// TwinCAT 3 PLC project MaterialHandling
// ProgramVersion: 3.1.4026.20
// CompilerDefines: VISU_USEPROPERTYINFO
// libraries:
//   Tc2_Standard, * (Beckhoff Automation GmbH)
//   Tc2_System, * (Beckhoff Automation GmbH)
// project tree:
//   Class Diagram/ Code Design Architecture.TcCD (not stored)
//   DUTs/ E_AutoState.TcDUT, E_ErrorHandling.TcDUT, E_Mode.TcDUT
//   / GlobalTextList.TcGTLO, PlcTask.TcTTO, Visualization Manager.TcVMO (not stored)
//   GVLs/ IOs.TcGVL
//   POUs/ FB_ErrorHandling.TcPOU, FB_AutoState.TcPOU, FB_ModeManager.TcPOU, MAIN.TcPOU, FB_StateMachine.TcPOU
//   VISUs/ Visualization.TcVIS
// real-time tasks:
//   TASK PlcTask: cycle T#10ms, priority 20, ADS port 350

CONFIGURATION MaterialHandling
    RESOURCE PLC ON TwinCAT3
        TASK PlcTask(INTERVAL := T#10ms, PRIORITY := 20);
        PROGRAM MAIN WITH PlcTask : MAIN;
    END_RESOURCE
END_CONFIGURATION

// ---- DUTs/E_AutoState.TcDUT
{attribute 'to_string'}
TYPE E_AutoState :
(
	Create_Product:= 10,
	Load_Conveyor:= 20,
	Transfer_To_MC:= 30,
	Machine_Start:= 40,
	Wait_Machine_Busy:= 50,
	Wait_Machine_Complete:= 60,
	Exit_MC:= 70,
	MOVE_To_Unload:= 80,
	Remove_Product:= 90,
	Complete:= 100
);
END_TYPE

// ---- DUTs/E_ErrorHandling.TcDUT
{attribute 'to_string'}
TYPE E_ErrorHandling :
(
	Fault := 900,
	Emergency := 999,
	No_Error := 0
);
END_TYPE

// ---- DUTs/E_Mode.TcDUT
{attribute 'to_string'}
TYPE E_Mode :
(
	Idle := 0,
	Auto := 1,
	Manual:= 2,
	Error:= 3
);
END_TYPE

// ---- GVLs/IOs.TcGVL
{attribute 'OPC.UA.DA' := '1'}
{attribute 'OPC.UA.DA.Access' := '3'}
VAR_GLOBAL
////////////////////////////////
    //Inputs...............
////////////////////////////////
(*1*)	 xSensor_LoadStation:        BOOL;
(*2*)    xSensor_BeforeEntry:        BOOL;
(*3*)    xSensor_AtExit:             BOOL;
(*4*)    xEStop:                     BOOL;    //Stop the complete Machine
(*5*)	 xPB_ManualRun_Pressed:      BOOL;    //PB = Push Button  
(*6*)    xMC_Opened:                 BOOL;    //MC = Machine Center
(*7*)    xMC_IsBusy:                 BOOL;
(*8*)	 xMC_HasError:               BOOL;
(*9*)    xrMC_Progress:              DINT;
(*10*)   xSel_Auto:                  BOOL;
(*11*)   xSel_Manual:                BOOL;
(*12*)	 xSel_OFF:                   BOOL;

(*13*)   xSystemPower:               BOOL;    // Power System ON/OFF - Input from HMI or Scene button
(*14*)   xSystemReset:               BOOL;    // System Reset - Input from HMI or Scene button 
/////////////////////////////////
    //Outputs...............
/////////////////////////////////
(*1*)	 xEmitter:                   BOOL;
(*2*)    xConv_LoadStation:          BOOL;    //Conv = Conveyor
(*3*)    xCurvedConv_CCW:            BOOL;
(*4*)    xConv_BeforeEntry:          BOOL;    //Stop the complete Machine
(*5*)	 xMC_Start:                  BOOL;    //PB = Push Button
(*6*)    xMC_Stop:                   BOOL;    //MC = Machine Center
(*7*)    xMC_Reset:                  BOOL;
(*8*)	 xMC_ProduceLids:            BOOL;    //True: Produce Lids , False: Produce Bases
(*9*)    xConv_AfterProcess:         BOOL;
(*10*)   xRemover:                   BOOL;
(*11*)   xPb_ManualRun_Light:        BOOL;
END_VAR

// ---- POUs/MAIN.TcPOU
PROGRAM MAIN
VAR
	fbStateMachine: FB_StateMachine;
	eErrorType: E_ErrorHandling;
	xEmitter_Manual: BOOL;  //Simulation
	eMode: E_Mode;
	////// Inputs & Outputs
	xEStop: BOOL;
	xPB_ManualRun_Pressed: BOOL;
	xSel_Auto: BOOL;
    xSel_Manual: BOOL;
	///////////
	xEmitter: BOOL;
	xConv_LoadStation: BOOL;
	xCurvedConv_CCW: BOOL;
	xConv_BeforeEntry: BOOL;
	xMC_Start: BOOL;
	xMC_Stop: BOOL;
	xMC_Reset: BOOL;
	xMC_ProduceLids: BOOL;
	xConv_AfterProcess: BOOL;
	xRemover: BOOL;
END_VAR


xEStop:= NOT IOs.xEStop;
xPB_ManualRun_Pressed:= IOs.xPB_ManualRun_Pressed;
xSel_Auto:= IOs.xSel_Auto;
xSel_Manual:= IOs.xSel_Manual;

IF IOs.xSystemPower THEN
	fbStateMachine(xEmitter_Manual:= xEmitter_Manual,xESTOP:= xESTOP, xPB_ManualRun_Pressed:= xPB_ManualRun_Pressed, xSel_Auto:= xSel_Auto, xSel_Manual:= xSel_Manual);
    eMode := fbStateMachine.eMode;
    eErrorType:= fbStateMachine.eErrorType;
END_IF


IOs.xEmitter := fbStateMachine.xEmitter;
IOs.xConv_LoadStation := fbStateMachine.xConv_LoadStation;
IOs.xCurvedConv_CCW := fbStateMachine.xCurvedConv_CCW;
IOs.xConv_BeforeEntry := fbStateMachine.xConv_BeforeEntry;
IOs.xMC_Start := fbStateMachine.xMC_Start;
IOs.xMC_Stop := fbStateMachine.xMC_Stop;
IOs.xMC_Reset := fbStateMachine.xMC_Reset;
IOs.xMC_ProduceLids := fbStateMachine.xMC_ProduceLids;
IOS.xConv_AfterProcess := fbStateMachine.xConv_AfterProcess; 
IOs.xRemover := fbStateMachine.xRemover;

END_PROGRAM

// ---- POUs/FB_StateMachine.TcPOU
FUNCTION_BLOCK FB_StateMachine

VAR
	fbModeManager: FB_ModeManager;
	fbAutoState: FB_AutoState;
	xEnable_Auto: BOOL;
	xReset_Auto: BOOL;
END_VAR
VAR_INPUT
	xEmitter_Manual: BOOL;
	xEStop: BOOL;
	xPB_ManualRun_Pressed: BOOL;
	xSel_Auto: BOOL;
    xSel_Manual: BOOL;
END_VAR
VAR_OUTPUT
	eErrorType: E_ErrorHandling;
	eMode: E_Mode;
	
	xEmitter: BOOL;
	xConv_LoadStation: BOOL;
	xCurvedConv_CCW: BOOL;
	xConv_BeforeEntry: BOOL;
	xMC_Start: BOOL;
	xMC_Stop: BOOL;
	xMC_Reset: BOOL;
	xMC_ProduceLids: BOOL;
	xConv_AfterProcess: BOOL;
	xRemover: BOOL;
END_VAR

fbModeManager(xEStop := xEStop, xSel_Auto:= xSel_Auto, xSel_Manual:= xSel_Manual);
eMode := fbModeManager.eMode;
eErrorType:= fbModeManager.eErrorType;

IF eMode = Auto THEN
	xEnable_Auto := TRUE;
	xReset_Auto := FALSE;
END_IF
IF eMode = Idle OR eMode = Manual THEN
		xEnable_Auto := FALSE;
	    xReset_Auto := TRUE;
END_IF
	
 CASE eMode OF
	
	Auto:
	   
	   fbAutoState(xEnable:=xEnable_Auto, xReset:=xReset_Auto);
	   
	   xEmitter := fbAutoState.xEmitter;
       xConv_LoadStation := fbAutoState.xConv_LoadStation;
	   xCurvedConv_CCW := fbAutoState.xCurvedConv_CCW;
	   xConv_BeforeEntry := fbAutoState.xConv_BeforeEntry;
	   xMC_Start := fbAutoState.xMC_Start;
	   xMC_ProduceLids := fbAutoState.xMC_ProduceLids;
	   xConv_AfterProcess := fbAutoState.xConv_AfterProcess;
	   xRemover := fbAutoState.xRemover;
	   
	Manual:
	   
	   IF xPB_ManualRun_Pressed THEN
		   xMC_Start := xPB_ManualRun_Pressed;  //Robot in the Scene is predefined to work only when the raw material detected from the cell-Sensor; IF operator released the PB during the Transfer, it supposed to finish the current job unless he pressed Stop
           //xPb_ManualRun_Light:= TRUE;    don't forget
		   xConv_LoadStation:= TRUE;
		   xCurvedConv_CCW:= TRUE;
		   xConv_BeforeEntry:= TRUE;
		   xConv_AfterProcess:=TRUE;
		   xEmitter := xEmitter_Manual;  //Operator should feed the Material manually obe by one (Later with HMI)
		   xRemover:= TRUE;
	   END_IF
	   
	   fbAutoState(xEnable:=xEnable_Auto, xReset:=xReset_Auto);
	  	
	 Idle:
	    
	    xConv_LoadStation:= FALSE;
		xCurvedConv_CCW:= FALSE;
		xConv_BeforeEntry:= FALSE;
		xConv_AfterProcess:= FALSE;
		xMC_Start:= FALSE;
		xMC_Stop:= FALSE;
		xEmitter:= FALSE;
		xRemover:= FALSE;
		xMC_Reset:= TRUE;
		xMC_Reset:= FALSE; //Trigger once at the beginning
		
		fbAutoState(xEnable:=xEnable_Auto, xReset:=xReset_Auto);
	  
  END_CASE

END_FUNCTION_BLOCK

// ---- POUs/FB_ModeManager.TcPOU
FUNCTION_BLOCK FB_ModeManager
VAR_INPUT
	xEStop: BOOL;
	xSel_Auto: BOOL;
	xSel_Manual: BOOL;
END_VAR
VAR_OUTPUT
	eMode: E_MODE;
	eErrorType: E_ErrorHAndling;
END_VAR
VAR
	fbErrorHandling: FB_ErrorHAndling;
END_VAR

IF IOs.xMC_HasError OR xEStop THEN  //Emergency_Stop is NC designed!
	eMode:= Error;
  ELSIF IOs.xSel_Auto THEN
   eMode:= Auto;
	ELSIF IOs.xSel_Manual THEN
		eMode:= Manual;
		ELSE
			eMode:= Idle;
END_IF


fbErrorHandling(xEStop := xEStop);
eErrorType:= fbErrorHandling.eErrorHandling;

END_FUNCTION_BLOCK

// ---- POUs/FB_ErrorHandling.TcPOU
FUNCTION_BLOCK FB_ErrorHandling
VAR_INPUT
	xEStop: BOOL;
END_VAR
VAR_OUTPUT
	eErrorHandling: E_ErrorHandling;
END_VAR
VAR
END_VAR

IF xEStop THEN
	eErrorHandling:= Emergency;
ELSIF IOs.xMC_HasError THEN
		eErrorHandling:= Fault;
		ELSE
			eErrorHandling:= No_Error;
END_IF

END_FUNCTION_BLOCK

// ---- POUs/FB_AutoState.TcPOU
FUNCTION_BLOCK FB_AutoState

VAR
	eAutoState: E_AutoState := Create_Product;
	//pPointer: POINTER TO E_MODE;
END_VAR
VAR_INPUT
	xEnable: BOOL;
	xReset: BOOL;
END_VAR
VAR_OUTPUT
	xEmitter: BOOL;
	xConv_LoadStation: BOOL;
	xCurvedConv_CCW: BOOL;
	xConv_BeforeEntry: BOOL;
	xMC_Start: BOOL;
	xMC_ProduceLids: BOOL;
	xConv_AfterProcess: BOOL;
	xRemover: BOOL;
END_VAR

IF xReset THEN
	IF IOs.xSystemReset THEN  //If Operator clicked reset=> Product on conveyor has been cleared ; If Not => system will continue running same product when back to Auto 
     eAutoState:= Create_Product;
    END_IF
   ELSIF xEnable THEN	
	
CASE eAutoState OF

(*10*) Create_Product:
	
	   xEmitter:= TRUE;
	   IF IOs.xSensor_LoadStation THEN
		  eAutoState := Load_Conveyor;
	   END_IF
	
(*20*) Load_Conveyor: 
	
	   xEmitter := FALSE;
	   xConv_LoadStation:= TRUE;
	   IF NOT IOs.xSensor_LoadStation THEN
		   eAutoState:= Transfer_To_MC;
	   END_IF
 
(*30*) Transfer_To_MC: 
	
	   xCurvedConv_CCW:= TRUE;
	   xConv_BeforeEntry:= TRUE;
	   IF IOs.xSensor_BeforeEntry THEN
		   eAutoState:= Machine_Start;
	   END_IF
	   
(*40*) Machine_Start: 

       xConv_LoadStation:= FALSE;
       xCurvedConv_CCW:= FALSE;
       xMC_Start:= TRUE;
       xMC_ProduceLids:= 0; //0 Produce base
	   IF IOs.xMC_IsBusy THEN
       eAutoState:= Wait_Machine_Busy;
	   END_IF
	   
(*50*) Wait_Machine_Busy: 
	 
	    xConv_BeforeEntry:= FALSE;
		IF (IOs.xrMC_Progress > 0) AND (IOs.xrMC_Progress < 100) THEN
		eAutoState:= Wait_Machine_Complete;
	    END_IF
	 
(*60*) Wait_Machine_Complete:  
	   
	   xMC_Start:= FALSE;
	   IF NOT (IOs.xMC_IsBusy AND IOs.xMC_HasError) THEN  //It should get in this State after checking outside no errors, should be considered here again ??
		   
		   eAutoState:= Exit_MC;
	   END_IF
	   
(*70*) Exit_MC:  
	   
	   xConv_AfterProcess:= TRUE;
	   eAutoState:= Move_To_Unload;
	   
(*80*)  MOVE_To_Unload: 
	 
	   IF IOs.xSensor_AtExit THEN
		   eAutoState:= Remove_Product;
	   END_IF
	   	 
(*90*)  Remove_Product: 
	 
			xRemover:= TRUE;
			eAutoState:= Complete;
					
(*100*) Complete:  
	 
		IF NOT IOs.xSensor_AtExit THEN
			xConv_AfterProcess:= FALSE;
			xRemover:= FALSE;
			eAutoState:= Create_Product;
		END_IF
	 
END_CASE
END_IF

END_FUNCTION_BLOCK

// ---- GlobalTextList.TcGTLO
TEXTLIST GlobalTextList
  116 = 'Power ON'
  152 = 'Reset'
  297 = 'Run'
  612 = 'Scene (Reset)'
  12 = 'Scene (Run)'
  870 = 'Scene Reset'
  21 = 'System Reset'
END_TEXTLIST

// ---- VISUs/Visualization.TcVIS
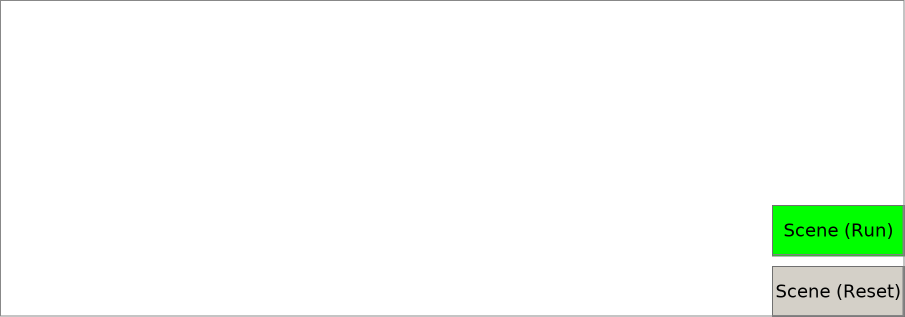
VISUALIZATION Visualization  // 905x317
    Button (772,205 133x51), "Scene (Run)"
        toggle xSystemPower
    Button (772,266 133x51), "Scene (Reset)"
        tap xSystemReset
END_VISUALIZATION
